# EPICS autosave request: 100idPyCRLApp/Db/slitTestTools_settings.req
$(P)$(SLITH).VAL
$(P)$(SLITV).VAL
